TYPE ST_AFS60_Cam :
STRUCT
	bEnable				: BOOL;
	nLowerLimit1		: UDINT;
	nLowerLimit2		: UDINT;
	nUpperLimit1		: UDINT;
	nUpperLimit2		: UDINT;
END_STRUCT
END_TYPE

(* stored: Version 1.1.0.1, ProductVersion 3.1.4024.15
   DUT ST_AFS60_Cam: Id {48b24227-87dc-458f-ab80-1056987bff47} *)
